TYPE ST_ExtractiveOnOffValveValues :
STRUCT
	open : BOOL;
END_STRUCT
END_TYPE

(* stored: Version 1.1.0.1, ProductVersion 3.1.4024.9
   DUT ST_ExtractiveOnOffValveValues: Id {45d9709c-00d9-43c5-be85-060be4de78ac} *)
